// TwinCAT 3 PLC project Untitled1
// ProgramVersion: 3.1.4022.3
// libraries:
//   Tc2_Standard, * (Beckhoff Automation GmbH)
//   Tc2_System, * (Beckhoff Automation GmbH)
//   Tc3_EventLogger, * (Beckhoff Automation GmbH)
//   Tc3_Module, * (Beckhoff Automation GmbH)
// project tree:
//   / PlcTask.TcTTO
//   POUs/ MAIN.TcPOU
// real-time tasks:
//   TASK PlcTask: cycle T#10ms, priority 20, ADS port 350

CONFIGURATION Untitled1
    RESOURCE PLC ON TwinCAT3
        TASK PlcTask(INTERVAL := T#10ms, PRIORITY := 20);
        PROGRAM MAIN WITH PlcTask : MAIN;
    END_RESOURCE
END_CONFIGURATION

// ---- POUs/MAIN.TcPOU
PROGRAM MAIN
VAR
	xCreateEvents		:BOOL:=TRUE; //Init
	
	xRaiseAllEvents		:BOOL;
	
	xRaiseTempAlarm		:BOOL;
	xConfirmTempAlarm	:BOOL;
	xClearTempAlarm		:BOOL;
	fTemp				:LREAL;
	fbAlarmTempToHigh	:FB_TcAlarm;
	eConfirmationState	:TcEventConfirmationState;
	
	xRaiseAlarm1		:BOOL;
	xConfirmAlarm1		:BOOL;
	xClearAlarm1		:BOOL;
	fbAlarm1			:FB_TcAlarm;

	xRaiseAlarm2		:BOOL;
	xConfirmAlarm2		:BOOL;
	xClearAlarm2		:BOOL;
	fbAlarm2			:FB_TcAlarm;
	
	xRaiseAlarm3		:BOOL;
	xConfirmAlarm3		:BOOL;
	xClearAlarm3		:BOOL;
	fbAlarm3			:FB_TcAlarm;
	
	fbTcEventLogger		:FB_TcEventLogger;
	xConfirm			: BOOL;
	xClear				: BOOL;
	
	
	tonSendInternal		:TON;
	xSendMsg			:BOOL;
	iCounter			:UDINT;
	fbMsgHelloWorld		:FB_TcMessage;
	

END_VAR

//Init - Create the events
IF xCreateEvents THEN
	xCreateEvents:=FALSE;
	
	fbAlarmTempToHigh.CreateEx(TC_EVENTS.Machine_XYZ.TempToHigh,1,0);
	
	fbAlarm1.CreateEx(TC_EVENTS.Machine_XYZ.Alarm_1,1,0);
	
	fbAlarm2.CreateEx(TC_EVENTS.Machine_XYZ.Alarm_2,1,0);
	
	fbAlarm3.CreateEx(TC_EVENTS.Machine_XYZ.Alarm_3,1,0);
	
	fbMsgHelloWorld.CreateEx(TC_EVENTS.Machine_XYZ.HelloWorldMsg,0);	
END_IF

//Raise all events
IF xRaiseAllEvents THEN
	xRaiseAllEvents:=FALSE;
	xRaiseAlarm1:=TRUE;
	xRaiseAlarm2:=TRUE;
	xRaiseAlarm3:=TRUE;
	xRaiseTempAlarm:=TRUE;
	xSendMsg:=TRUE;
END_IF

//Temp Alarm
IF xRaiseTempAlarm  THEN
	xRaiseTempAlarm:=FALSE;
	fTemp:=fTemp+10;
	fbAlarmTempToHigh.ipArguments.Clear().AddLReal(fTemp);
	fbAlarmTempToHigh.Raise(0);
END_IF
IF xConfirmTempAlarm THEN
	xConfirmTempAlarm:=FALSE;
	fbAlarmTempToHigh.Confirm(0);
END_IF
IF xClearTempAlarm THEN
	xClearTempAlarm:=FALSE;
	fbAlarmTempToHigh.Clear(0,0);
END_IF

//Alarm 1
IF xRaiseAlarm1 THEN
	xRaiseAlarm1:=FALSE;
	fbAlarm1.Raise(0);
END_IF
IF xConfirmAlarm1 THEN
	xConfirmAlarm1:=FALSE;
	fbAlarm1.Confirm(0);
END_IF
IF xClearAlarm1 THEN
	xClearAlarm1:=FALSE;
	fbAlarm1.Clear(0,0);
END_IF

//Alarm 2
IF xRaiseAlarm2 THEN
	xRaiseAlarm2:=FALSE;
	fbAlarm2.Raise(0);
END_IF
IF xConfirmAlarm2 THEN
	xConfirmAlarm2:=FALSE;
	fbAlarm2.Confirm(0);
END_IF
IF xClearAlarm2 THEN
	xClearAlarm2:=FALSE;
	fbAlarm2.Clear(0,0);
END_IF

//Alarm 3
IF xRaiseAlarm3 THEN
	xRaiseAlarm3:=FALSE;
	fbAlarm3.Raise(0);
END_IF
IF xConfirmAlarm3 THEN
	xConfirmAlarm3:=FALSE;
	fbAlarm3.Confirm(0);
END_IF
IF xClearAlarm3 THEN
	xClearAlarm3:=FALSE;
	fbAlarm3.Clear(0,0);
END_IF



//Confirm and clear all alarms
IF xConfirm THEN
	xConfirm:=FALSE;
	fbTcEventLogger.ConfirmAllAlarms(0);
END_IF
IF xClear THEN
	xClear:=FALSE;
	fbTcEventLogger.ClearAllAlarms(0,0);
END_IF

	eConfirmationState:=fbAlarmTempToHigh.eConfirmationState;

//Message
IF xSendMsg THEN
	xSendMsg:=FALSE;
	iCounter:=iCounter+1;
	fbMsgHelloWorld.ipArguments.Clear().AddUDInt(iCounter);
	fbMsgHelloWorld.Send(0);
END_IF

END_PROGRAM
